// TIA Portal V20 export
DATA_BLOCK "Side_MOVIKIT"   // DB18
{ S7_Optimized_Access := 'TRUE' }
// stored: MemoryReserve 0
   VAR
      S2_R1_PI : "SEW_MOVIKIT_VelocityDrive_STATUS_V2.1";
      S2_R1_PO : "SEW_MOVIKIT_VelocityDrive_SETPOINTS_V2.1";
      S2_R2_PI : "SEW_MOVIKIT_VelocityDrive_STATUS_V2.1";
      S2_R2_PO : "SEW_MOVIKIT_VelocityDrive_SETPOINTS_V2.1";
      S2_R1_Communication_OK { S7_SetPoint := 'True'} : Bool;
      S2_R2_Communication_OK { S7_SetPoint := 'True'} : Bool;
      S1_R1_PI : "SEW_MOVIKIT_VelocityDrive_STATUS_V2.1";
      S1_R1_PO : "SEW_MOVIKIT_VelocityDrive_SETPOINTS_V2.1";
      S1_R2_PI : "SEW_MOVIKIT_VelocityDrive_STATUS_V2.1";
      S1_R2_PO : "SEW_MOVIKIT_VelocityDrive_SETPOINTS_V2.1";
      S1_R1_Communication_OK { S7_SetPoint := 'True'} : Bool;
      S1_R2_Communication_OK { S7_SetPoint := 'True'} : Bool;
   END_VAR
BEGIN
END_DATA_BLOCK
